{attribute 'OPC.UA.DA' := '1'}
FUNCTION_BLOCK DM430GNScreenFS EXTENDS DM430GNScreen
VAR_INPUT
END_VAR
VAR_OUTPUT
END_VAR
VAR
	{attribute 'OPC.UA.DA' := '0'}
	_config : DM430GNScreenConfig;
	{attribute 'OPC.UA.DA' := '0'}
	_coeAccess : CoeAccess;
	{attribute 'OPC.UA.DA' := '0'}
	_initConfigSerialCom : BOOL;
	{attribute 'OPC.UA.DA' := '0'}	
	_serialCom  : SerialCom(Prefix :='', Suffix := Const.CARRIAGE_RETURN);
	{attribute 'OPC.UA.DA' := '0'}
	_refSerialCom : REFERENCE TO SerialCom(Prefix :='', Suffix := Const.CARRIAGE_RETURN) := _serialCom;	
	
	{attribute 'OPC.UA.DA' := '0'}
	_pulseGeneratorInit : TON;	
	{attribute 'OPC.UA.DA' := '0'}
	_itemInit : INT;
END_VAR

IF _config.IsSimulated THEN
	SUPER^(Conf := _config, SerialCom := _serialCom, RefSerialCom := _refSerialCom);
ELSE
	IF NOT InitConfigSerialCom THEN
		ConfigureSerialCom();
	ELSIF THIS^.Status = TExecutionState.Ready THEN
		IF _refSerialCom.ErrorReceiveId = COMERROR_NOERROR THEN
			_refSerialCom(TxBuffer:= HardwareGlobalVariables.TxBufferDM430GNScreenFS, 
						  RxBuffer:= HardwareGlobalVariables.RxBufferDM430GNScreenFS);
		END_IF						  			
					
		SUPER^(Conf := _config, SerialCom := _serialCom, RefSerialCom := _refSerialCom);

		// Init device
		InitDevice(); 			
	END_IF
END_IF

METHOD ConfigureSerialCom
VAR_INPUT
END_VAR

VAR
	Status: INT;
END_VAR
IF _coeAccess.CoeOperation.Ready THEN
	_logger.Information(_message.Reset().Append('Start configuration com serial').ToString());
END_IF;	

_coeAccess.CoeOperation.Start();
_coeAccess(SerialCommunication := _config.SerialCommunication);
	
IF _coeAccess.CoeOperation.Done THEN
	_coeAccess.SetDone();
	
	_Logger.Information(_message.Reset().
							Append('{').Append(TO_STRING(THIS^.Family)).Append('} : ').
							Append(' - Status : ').Append(TO_STRING(_coeAccess.Status)).ToString());
	InitConfigSerialCom := TRUE;
END_IF
 
IF _coeAccess.CoeOperation.Error THEN	
	_coeAccess.SetError(0);
	
	_Logger.Error(_message.Reset().
							Append('{').Append(TO_STRING(THIS^.Family)).Append('} : ').
							Append(' - Status : ').Append(TO_STRING(_coeAccess.Status)).ToString());
	InitConfigSerialCom := TRUE;
END_IF

THIS^.Status := _coeAccess.Status;
State := _coeAccess.Status;
END_METHOD

METHOD FB_init : BOOL
VAR_INPUT
	bInitRetains : BOOL; // if TRUE, the retain variables are initialized (warm start / cold start)
	bInCopyCode : BOOL;  // if TRUE, the instance afterwards gets moved into the copy code (online change)
	Config : DM430GNScreenConfig;
END_VAR
IF Config.IsEnabled THEN
	_config := Config;
	
	SUPER^._screenConfig.Name := Config.Name;
	SUPER^._screenConfig.DeviceID := Config.DeviceID;
	SUPER^._screenConfig.IsEnabled := Config.IsEnabled;
	SUPER^._screenConfig.LogLevel := Config.LogLevel;
	
	SUPER^.Name := Config.Name;
	SUPER^.DeviceID := Config.DeviceID;	
	THIS^.Family := DeviceFamily.Screen;
		
	_Logger.Information(_message.Reset().Append('Init ').
							Append('{').Append(TO_STRING(THIS^.Family)).Append('} - ').
							Append('{').Append(TO_STRING(Config.Name)).Append('}').ToString());																													
END_IF
END_METHOD

PROPERTY InitConfigSerialCom : BOOL
GET
InitConfigSerialCom := _initConfigSerialCom;
END_GET
SET
_initConfigSerialCom := InitConfigSerialCom;
END_SET
END_PROPERTY

METHOD InitDevice
VAR_INPUT
END_VAR
VAR	
END_VAR
IF NOT _initDevice THEN		
	IF _pulseGeneratorInit.Q THEN
		_pulseGeneratorInit(IN := FALSE, PT := T#10MS);
			
		CASE _itemInit OF
			0:  _logger.Information(_message.Reset().Append(_config.Name).Append(' - Start to on').ToString());		
				_itemInit := 1;
				
			1:  _initDevice := TRUE;
				_itemInit := 0;
		END_CASE
	ELSE
		_pulseGeneratorInit(IN := TRUE, PT := T#500MS);	
	END_IF
END_IF
END_METHOD

END_FUNCTION_BLOCK

(* stored: Version 1.1.0.1, ProductVersion 3.1.4024.12
   POU DM430GNScreenFS: Id {30925906-f928-42db-ad44-bfdf9446b57f}, SpecialFunc None
   Folder Commands: Id {0812b7c2-1ae7-447a-9d38-fca7412a7f3a}
   Method ConfigureSerialCom: Id {9e22e0e1-2520-4d6c-a85c-66636ebe9d8b}
   Method FB_init: Id {e43734c5-fc03-4d0c-9616-def70286f00c}
   Property InitConfigSerialCom: Id {c9bdc576-f2be-4a0f-b7c3-7d1ca4fb9c39}
   Get Get: Id {3f19747e-e6d7-4ec1-b2d2-820fd55e3cea}
   Set Set: Id {f7ab7a19-6a58-42a8-85fd-2b324faa5f8e}
   Method InitDevice: Id {e4b4a045-3dd2-4739-8f51-a2e706adfa48} *)
